SUBAPPLICATION NumericValue_TO_AR2 (* VT-Eingabefeld (CInputNumber) lesen und als AR2 (bidirektional) an einen Consumer weiterreichen (z.B. AR_CALIBRATE_SQ_REF.Y_Offset/.Y_Scale, oder direkt an ein INI_AR2). Speichert NICHT selbst - der Consumer persistiert (z.B. via ZERO/SPAN+INI_AR2), das Echo kommt hier ueber denselben AR2-Plug zurueck und wird auf das VT-Feld zurueckgeschrieben (auch beim Boot) *)
  (* Standard: 61499-2; Description: Copyright (c) 2026 Meisterschulen am Ostbahnhof This program and the accompanying materials are made available under the terms of the Eclipse Public License 2.0 which is available at https://www.eclipse.org/legal/epl-2.0/ SPDX-License-Identifier: EPL-2.0 *)
  (* Version 1.0, 2026-08-31, Franz Höpfinger, Meisterschulen am Ostbahnhof, Renamed from INI_IN_AND_STORE_AR2 - this SubApp is a pure VT-to-AR2 bridge, it does not persist anything itself *)
  PACKAGE MyLib::sys;
  IMPORT isobus::UT::Q::const::IDs::ID_NULL;
  IMPORT logiBUS::utils::conversion::phys::NumericObjectPool_S;
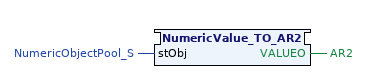
  VAR_INPUT
    stObj : logiBUS::utils::conversion::phys::NumericObjectPool_S := (u16ObjId := ID_NULL, r32Scale := 1.0, i32Offset := 0, u8Decimals := 0);
  END_VAR
  PLUGS
    VALUEO : adapter::types::bidirectional::AR2;
  END_PLUGS
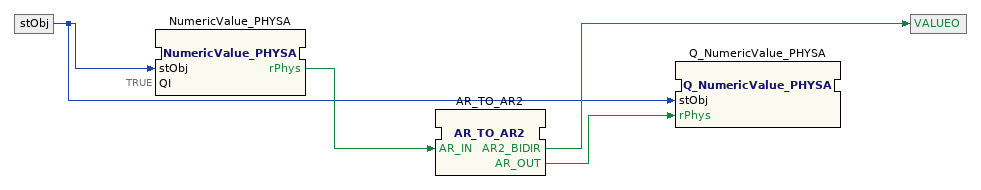
  FBS
    NumericValue_PHYSA : isobus::UT::io::NumericValue::NumericValue_PHYSA(QI := TRUE);
    AR_TO_AR2 : adapter::conversion::bidirectional::AR_TO_AR2;
    Q_NumericValue_PHYSA : isobus::UT::Q::Q_NumericValue_PHYSA;
  END_FBS
  DATA_CONNECTIONS
    stObj TO Q_NumericValue_PHYSA.stObj;
    stObj TO NumericValue_PHYSA.stObj;
  END_CONNECTIONS
  ADAPTER_CONNECTIONS
    NumericValue_PHYSA.rPhys TO AR_TO_AR2.AR_IN;
    AR_TO_AR2.AR2_BIDIR TO VALUEO;
    AR_TO_AR2.AR_OUT TO Q_NumericValue_PHYSA.rPhys;
  END_CONNECTIONS
END_SUBAPPLICATION
